// TIA Portal V17 export
// export: Created 2023-12-22T15:03:09.7524479Z, ExportSetting WithDefaults, DisplayName Totally Integrated Automation Portal, DisplayVersion V17, DisplayName TIA Portal Openness, DisplayVersion V17, DisplayName TIA Portal Version Control Interface, DisplayVersion V17, DisplayName STEP 7 Professional, DisplayVersion V17, DisplayName STEP 7 Safety, DisplayVersion V17, DisplayName WinCC Advanced, DisplayVersion V17
DATA_BLOCK "PE_DB"   // DB397
{ S7_Optimized_Access := 'FALSE' }
VERSION : 0.1
// stored: AutoNumber false, DBAccessibleFromOPCUA true, DBAccessibleFromWebserver true, IsOnlyStoredInLoadMemory false, IsWriteProtectedInAS false
   VAR RETAIN
      PE : Array[0..20] of Struct   // Чтение - Input Register (04), Запись - Holding Register (06)
         PE : Real;   // Накопленный объем +
         res_0 : Real;   // Накопленный объём -
         res_1 : Real;   // Мгновенный расход
         res_2 : Real;   // Температура канала 1, С
         res_3 : Real;   // Температура канала 2, С
         res_4 : Real;   // Давление среды, кПа
         Use { S7_SetPoint := 'True'} : Bool;
         Link : Bool;
         NoRead : Bool;
         NoWrite : Bool;
         ID { S7_SetPoint := 'True'} : Int;
         ADDR { S7_SetPoint := 'True'} : UInt;
         "Name" { S7_SetPoint := 'True'} : String[10];
      END_STRUCT;
   END_VAR
BEGIN
   PE[0].Use := FALSE;
   PE[1..2].Use := TRUE;
   PE[3..10].Use := FALSE;
   PE[0].ID := 0;
   PE[1..2].ID := 14;
   PE[3..10].ID := 0;
   PE[0].ADDR := 0;
   PE[1].ADDR := 41;
   PE[2].ADDR := 42;
   PE[3..10].ADDR := 0;
   PE[0]."Name" := '';
   PE[1]."Name" := 'FE';
   PE[2..10]."Name" := '';
END_DATA_BLOCK
